FUNCTION_BLOCK SKILL_FailMerge (* Merges two failure events with their error codes into one *)
  (* Standard: 61499-2 *)
  (* Version 0.1, 2026-09-28, Project contributors, AAU Smart Production Lab *)
  PACKAGE modlib;
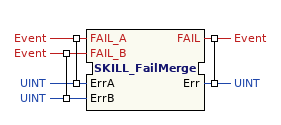
  EVENT_INPUT
    FAIL_A WITH ErrA;
    FAIL_B WITH ErrB;
  END_EVENT
  EVENT_OUTPUT
    FAIL WITH Err;
  END_EVENT
  VAR_INPUT
    ErrA : UINT;
    ErrB : UINT;
  END_VAR
  VAR_OUTPUT
    Err : UINT;
  END_VAR
  EC_STATES
    FAIL_A : FAIL_A -> FAIL;
    FAIL_B : FAIL_B -> FAIL;
  END_STATES
  ALGORITHM FAIL_A IN ST:
Err := ErrA;
  END_ALGORITHM
  ALGORITHM FAIL_B IN ST:
Err := ErrB;
  END_ALGORITHM
END_FUNCTION_BLOCK
